FUNCTION_BLOCK RampLimitFS (* Setpoint Ramp: Step up and down Values with Fast and Slow mode *)
  (* Standard: 61499-1; Description: Copyright (c) 2024 HR Agrartechnik GmbH This program and the accompanying materials are made available under the terms of the Eclipse Public License 2.0 which is available at https://www.eclipse.org/legal/epl-2.0/ SPDX-License-Identifier: EPL-2.0 Setpoint Ramp: Step up and down Values, like well-known for the cruise control in your Car. Long press increase or decrease by 10, short press increase or decrease at 1. this FB adds Maximum and Minimum Value and also Inputs to set them. For some Applications it is neccessary to store the setpoint in Non-Volatile Storage, e.g. with a ini File, for this we have here a LOAD event input which loads value from the PV input *)
  (* Version 1.0, 2024-09-20, Franz Höpfinger, HR Agrartechnik GmbH *)
  (* Version 1.1, 2024-10-02, Franz Höpfinger, HR Agrartechnik GmbH, Rename to RampLimitFS *)
  (* Version 3.0, 2025-04-14, Patrick Aigner, changed package *)
  PACKAGE eclipse4diac::signalprocessing;
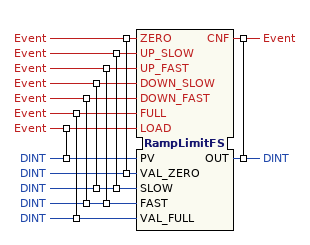
  EVENT_INPUT
    ZERO WITH VAL_ZERO; (* Set OUT to VAL_ZERO *)
    UP_SLOW WITH SLOW; (* Increase OUT by SLOW *)
    UP_FAST WITH FAST; (* Increase OUT by FAST *)
    DOWN_SLOW WITH SLOW; (* Decrease OUT by SLOW *)
    DOWN_FAST WITH FAST; (* Decrease OUT by FAST *)
    FULL WITH VAL_FULL; (* Set OUT to VAL_FULL *)
    LOAD WITH PV; (* Load PV into OUT *)
  END_EVENT
  EVENT_OUTPUT
    CNF WITH OUT; (* Execution Confirmation *)
  END_EVENT
  VAR_INPUT
    PV : DINT; (* Preset Value *)
    VAL_ZERO : DINT; (* Minimum Value *)
    SLOW : DINT; (* Value for slower Change *)
    FAST : DINT; (* Value for faster change *)
    VAL_FULL : DINT; (* Maximum Value *)
  END_VAR
  VAR_OUTPUT
    OUT : DINT; (* Output *)
  END_VAR
  ALGORITHM ZERO IN ST:
OUT := VAL_ZERO;
  END_ALGORITHM
  ALGORITHM UP_SLOW IN ST:
OUT := ADD(OUT, SLOW);
IF GT(OUT, VAL_FULL) THEN
	OUT := VAL_FULL;
END_IF;
  END_ALGORITHM
  ALGORITHM UP_FAST IN ST:
OUT := ADD(OUT, FAST);
IF GT(OUT, VAL_FULL) THEN
	OUT := VAL_FULL;
END_IF;
  END_ALGORITHM
  ALGORITHM DOWN_SLOW IN ST:
OUT := SUB(OUT, SLOW);
IF LT(OUT, VAL_ZERO) THEN
	OUT := VAL_ZERO;
END_IF;
  END_ALGORITHM
  ALGORITHM DOWN_FAST IN ST:
OUT := SUB(OUT, FAST);
IF LT(OUT, VAL_ZERO) THEN
	OUT := VAL_ZERO;
END_IF;
  END_ALGORITHM
  ALGORITHM FULL IN ST:
OUT := VAL_FULL;
  END_ALGORITHM
  ALGORITHM LOAD IN ST:
OUT := PV;
  END_ALGORITHM
END_FUNCTION_BLOCK
